													[(	byShrtAdr_Prim := 24, 
														byGrpAdr_Prim := 3, 
														eMod_Prim := E_DALIAddressType.Group, 
														byShrtAdr_Sec := 1, 
														byGrpAdr_Sec := 1, 
														//eMod_Sec := E_DALIAddressType.Short, 
														//byShrtAdr_Supl := 1,
														//eMod_Supl := E_DALIADDRESSTYPE.Group,
                                                        //byGrpAdr_Supl := 2, 
														DALI_LINE_NUM_PRIM := arrDALI_LINE_NUM_LIGHT[1], 
														DALI_LINE_NUM_SEC := 0, //0 = ingen zonestyring/vinduerække
														DALI_LINE_NUM_SUPL := arrDALI_LINE_NUM_PENDANTS[1]),
														
													(	byShrtAdr_Prim := 22, 
														byGrpAdr_Prim := 3, 
														eMod_Prim := E_DALIAddressType.Group, 
														byShrtAdr_Sec := 1, 
														byGrpAdr_Sec := 1, 
														//eMod_Sec := E_DALIAddressType.Short, 
														//byShrtAdr_Supl := 63, 
														DALI_LINE_NUM_PRIM := arrDALI_LINE_NUM_LIGHT[2], 
														DALI_LINE_NUM_SEC := 0, 
														DALI_LINE_NUM_SUPL := arrDALI_LINE_NUM_PENDANTS[2])];
														
	arrstLiveDataGruppe		: ARRAY [1..2] OF SH_Light.ST_LiveData;
	//stLiveData AT %MB22	: SH_Light.ST_LiveData;
	
	arrRunTuningGruppe: ARRAY[1..2] OF BOOL;
	
	bTopButtonZone1			: BOOL;
	bTopButtonZone1_Visu	: BOOL;
	bBottomButtonZone1		: BOOL;
	bBottomButtonZone1_Visu	: BOOL;
	bButtonZone2			: BOOL;
	bNeighborRoomsPir		: BOOL;
	fLuxOn					: REAL;
	fLuxDim					: REAL;
	tPIRDim					: TIME;
	tPIROff					: TIME;
	fOffsetSec				: REAL := 20;
	bOccupiedRoom			: BOOL;

	
// Sensor Settings
	//fbSensor					: SH_Light.FB_NIKO_P46xx_1Pcs;
	fbSensor					: SH_Light.FB_NIKO_P46xx_2Pcs;
	//bySensorAddr				: BYTE := x;
	arrSensorAddr				: ARRAY[1..2] OF BYTE := [3,4];
	bInitialize					: BOOL := TRUE;
	stDaliSensorSetup			: ST_DALI_NIKOP46SetupData := (
																nSensitivityPIRSegmentA := arrSensitivityOccupancy[1],
																nSensitivityPIRSegmentB := arrSensitivityOccupancy[2],
																nSensitivityPIRSegmentC := arrSensitivityOccupancy[3]);
	//bInitErr					: BOOL;
	//bInitDone					: BOOL;
	arrInitErr				: ARRAY [1..2] OF BOOL;
	arrInitDone				: ARRAY [1..2] OF BOOL;
	arrSensorScales				: ARRAY [1..10] OF SH_Light.ST_DALI_SensorScaleMode := [
																						(fMeassureMaxSensor := 1023, fReadMaxSensor := 1023),
																						(fMeassureMaxSensor := 1023, fReadMaxSensor := 1023),
																						8(())];
	bCancelHoldTimerOccupancy	: BOOL;
(*	eEventPriorityOccupancy		: E_DALIEventPriority := E_DALIEVENTPRIORITY.Middle;
	nHoldTimerOccupancy			: WORD := 5; // Value in s. 	
	nReportTimerOccupancy		: BYTE := 120; // Value in s, Preset manufacturer value
	nDeadtimeTimerOccupancy		: WORD := 100; // Value in ms, Predefined Value of DALI Standard
	bCancelHoldTimerOccupancy	: BOOL;
	nSensitivityOccupancy		: BYTE:= 3; //setting Sensivity (0..4) 0 (Off), 1 (Min), 2(Low), 3(High) and 4 (Max)

	bEnableLuxEvent				: BOOL;
	eEventPriorityBrightness	: E_DALIEventPriority := E_DALIEVENTPRIORITY.Middle;
	nDeadtimeTimerBrightness	: WORD := 1500; // Value in ms, Predefined Value of DALI Standard
	nHysteresisBrightness		: BYTE := 2; // Value in %
	nHysteresisMinBrightness	: BYTE := 10; // Absolute Value, depending on the manufacturer specific resolution
	nReportTimerBrightness		: BYTE := 120; // Value in s, Preset manufacturer value
*)

//ModbusComm setup
	
	fbWriteSPLuxLevel			: SH_Light.FB_TwoVal_SelectOne_RTrigChange;
	fbWritePirDelayTIme		: SH_Light.FB_TwoVal_SelectOne_RTrigChange;
	stRoomDataPLC				: SH_Light.ST_RoomDataPLC	:=	(
																	uiPirOffDelayTime	:= 30,
																	uiSpLuxLevel			:= 500,
																	uiPirDimDelayTime	:= 15,
																	uiSpDimLuxLevel		:= 200);
																	
	fbBallastOnHours			: SH_Light.FB_CountOnHours;
	bEnableHourCount			: BOOL := TRUE;
	
	//Non-persistent modbus data
	bPirActive_MB					AT%MX216.0	: BOOL;				//bPirLys i gammel kode
	uiActLuxLevel_MB			    AT%MB220		: UINT;				//intHMIAktueltLux i gammel kode
	uiActLightLevelPct_MB	        AT%MB224		: UINT;				//intDALI_Gruppe1_Lysniveau i gammel kode

	//For Conversion
	uiPirOffMinutes						: UINT;
	udTimeScaling						: UDINT := 60000;
	uiLuxOn								: UINT;
	
	//max values checks
	uiMaxLuxLevel						: UINT := 1023;
	uiMaxPirOffMinutes			     	: UINT := 180;
	
END_VAR

VAR CONSTANT
	//Sensor_DALI_LINE_NUM: BYTE := 3;
	Sensor_DALI_LINE_NUM				: BYTE := 2;
	arrDALI_LINE_NUM_LIGHT: ARRAY[1..2] OF BYTE := [1,2]; //korrekt rækkefølge nødvendig //rækkefølge og linje 
	arrDALI_LINE_NUM_PENDANTS: ARRAY[1..2] OF BYTE := [0,0]; //korrekt rækkefølge nødvendig. 0 = ingen pendler
	arrSensitivityOccupancy				: ARRAY[1..3] OF BYTE := [4,4,4];
END_VAR
VAR PERSISTENT
	stPirSensorData: SH_Light.ST_DALI_Sensor;
	arrstPirSensorDataLine: ARRAY[1..2] OF SH_Light.ST_DALI_Sensor; //hvad kan den her ??
	arrstTuneDataGruppe: ARRAY [1..2] OF SH_Light.ST_TuneData_EX;

	uiPirOffDelayTime_MB	AT%MB218	        : UINT;				//ntHMI_Pir_SetValue i gammel kode
	uiSPLuxLevel_MB			AT%MB222	   		: UINT;				//intHMI_Lux_SetValue i gammel kode
	uiBallastOnHours_MB		AT%MB226	        : UINT;		    	//dintHMILysbraendtimer1 i gammel kode
	byOnHoursOverflowCount			     		: BYTE;
END_VAR

A_Buttons();
A_LightCtrl();
A_Sensor();
A_ModbusComm();

ACTION A_Buttons:

bTopButtonZone1		:= bTopButtonZone1_Visu;
bBottomButtonZone1	:= bBottomButtonZone1_Visu;
END_ACTION

ACTION A_LightCtrl:
	

//gruppe 6
arrfbLysGruppe[1]( 
	nZoneID:= 1, 
	bButtonZone1:= bTopButtonZone1,
	bBottomButtonZone1 := bBottomButtonZone1, 
	bButtonZone2:= bButtonZone2,
	fLuxOn:= fLuxOn, 
	fLuxDim:= fLuxDim, 
	tPIRDim:= tPIRDim, 
	tPIROff:= tPIROff, 
	fOffsetSec:= fOffsetSec, 
	bReInit:= , 
	stDaliSetup:= arrstDaliSetupGruppe[1], 
	ipCommunication_Prim:= P_DALI_Background.arrfbKL6821Communication[arrDALI_LINE_NUM_LIGHT[1]], 
	//ipCommunication_Sec:= P_DALI_Background.arrfbKL6821Communication[arrDALI_LINE_NUM_LIGHT[1]], //samme som lyslinjen, hvis den ikke eksisterer
	//ipCommunication_Supl:= P_DALI_Background.arrfbKL6821Communication[arrDALI_LINE_NUM_LIGHT[1]],//samme som lyslinjen, hvis den ikke eksisterer 
	fMinOutputPowerLevelRoom:= 15, 
	fMaxOutputPowerLevelRoom:= 100, 
	nCycleTimeInMS:= SH_Light.DALI_Param.nPlcTaskCycleTimeInMS*nDimCmdCycleTimeFactor , 
	bRunTuning:= arrRunTuningGruppe[1], 
	bOccupiedRoom=> , 
	bError_Prim=> , 
	nError_Prim=> , 
	stTuneData:=arrstTuneDataGruppe[1] , 
	stPirSensorData:= stPirSensorData, 					//samme sensordata
	stLiveData:= arrstLiveDataGruppe[1]);

//gruppe 15	
arrfbLysGruppe[2]( 
	nZoneID:= 1, 
	bButtonZone1:= bTopButtonZone1,
	bBottomButtonZone1 := bBottomButtonZone1, 
	bButtonZone2:= bButtonZone2,
	fLuxOn:= fLuxOn, 
	fLuxDim:= fLuxDim, 
	tPIRDim:= tPIRDim, 
	tPIROff:= tPIROff, 
	fOffsetSec:= fOffsetSec, 
	bReInit:= , 
	stDaliSetup:= arrstDaliSetupGruppe[2], 
	ipCommunication_Prim:= P_DALI_Background.arrfbKL6821Communication[arrDALI_LINE_NUM_LIGHT[2]], 
	//ipCommunication_Sec:= P_DALI_Background.arrfbKL6821Communication[arrDALI_LINE_NUM_LIGHT[2]], //samme som lyslinjen, hvis den ikke eksisterer
	//ipCommunication_Supl:= P_DALI_Background.arrfbKL6821Communication[arrDALI_LINE_NUM_LIGHT[2]], //samme som lyslinjen, hvis den ikke eksisterer 
	fMinOutputPowerLevelRoom:= 15, 
	fMaxOutputPowerLevelRoom:= 100, 
	nCycleTimeInMS:= SH_Light.DALI_Param.nPlcTaskCycleTimeInMS*nDimCmdCycleTimeFactor , 
	bRunTuning:= arrRunTuningGruppe[2], 
	bOccupiedRoom=> , 
	bError_Prim=> , 
	nError_Prim=> , 
	stTuneData:=arrstTuneDataGruppe[2] , 
	stPirSensorData:= stPirSensorData, 					//samme sensordata
	stLiveData:= arrstLiveDataGruppe[2]);
END_ACTION

ACTION A_ModbusComm:
//Manage data for modbus communication

//Manage data for read-only in PLC
stRoomDataPLC.bPirActive			:= stPirSensorData.bPrc;
stRoomDataPLC.uiActLuxLevel			:= TO_UINT(TRUNC(stPirSensorData.fBrightness));
stRoomDataPLC.uiActLightLevelPct	:= TO_UINT(TRUNC(arrfbLysGruppe[1].fbBallast.fActlLgtLvl_Prim));
		//stRoomDataPLC.uiActLightLevelPct	:= TO_UINT(TRUNC(fbLys.fbBallast.fActlLgtLvl_Prim)); //if only one group light control
stRoomDataPLC.uiBallastOnHours		:= uiBallastOnHours_MB; //The calculation for BallastOnHours is stored directly to the MB register below


//Assign data for read-only to MB registers
bPirActive_MB			:= stRoomDataPLC.bPirActive;
uiActLuxLevel_MB		:= stRoomDataPLC.uiActLuxLevel;
uiActLightLevelPct_MB	:= stRoomDataPLC.uiActLightLevelPct;

	//calculate BallastOnHours
	fbBallastOnHours(
		bEnableHourCount	:= bEnableHourCount,
		bPauseCount			:= arrfbLysGruppe[1].fbLightCtrl.bOffZone1,
		uiOnHours			:= uiBallastOnHours_MB,			//OnHours is updated here
		byOverflowCount		:= byOnHoursOverflowCount);


//Manage data for read/write for both PLC and MB registers
fbWriteSPLuxLevel(	nMaxValOut	:= uiMaxLuxLevel,
					nValIn1		:= uiSPLuxLevel_MB,		//nValIn1 takes priotity in case of download or restart
					nValIn2		:= stRoomDataPLC.uiSpLuxLevel,
					nValOut		=> uiLuxOn
				);


fbWritePirDelayTIme(	nMaxValOut	:= uiMaxPirOffMinutes,
						nValIn1		:= uiPirOffDelayTime_MB,		//nValIn1 takes priotity in case of download or restart
						nValIn2		:= stRoomDataPLC.uiPirOffDelayTime,
						nValOut		=> uiPirOffMinutes
					);
					

//Convert read/write modbus data to appropriate datatypes in PLC
fLuxOn	:= TO_REAL(uiLuxOn);			
tPIROff	:= TO_TIME(uiPirOffMinutes*udTimeScaling); //Time conversion defaults to ms

fLuxDim	:= TO_REAL(stRoomDataPLC.uiSpDimLuxLevel);			
tPIRDim	:= TO_TIME(stRoomDataPLC.uiPirDimDelayTime*udTimeScaling); //Time conversion defaults to ms
END_ACTION

ACTION A_Sensor:

fbSensor.ipCommunication := P_DALI_Background.arrfbKL6821Communication[Sensor_DALI_LINE_NUM];

(*
fbSensor(
	byShrtAdr:= bySensorAddr,
	bInitialize:= bInitialize, 
	DALI_LINE_NUM:= Sensor_DALI_LINE_NUM, 
 	//bCancelHoldTimerOccupancy:= bCancelHoldTimerOccupancy, 
	stSensorSetup := stDaliSensorSetup,
	bInitErr=> bInitErr, 
	bInitDone=> bInitDone,
	stPirSensorData:= stPirSensorData, 
	arrSensorScales:= arrSensorScales);
*)

fbSensor(
	arrShrtAdr:= arrSensorAddr,
	bInitialize:= bInitialize, 
	DALI_LINE_NUM:= Sensor_DALI_LINE_NUM, 
 	//bCancelHoldTimerOccupancy:= bCancelHoldTimerOccupancy, 
	stSensorSetup := stDaliSensorSetup,
	arrInitErr=> arrInitErr, 
	arrInitDone=> arrInitDone,
	stPirSensorData:= stPirSensorData, 
	arrSensorScales:= arrSensorScales);
END_ACTION

END_PROGRAM

// ---- POUs/Alle_Rum/Trapper/P_Trappe_T5.TcPOU
PROGRAM P_Trappe_T5
VAR
	bDigitalPir				AT%I*	: BOOL;
	bTrappelysNC		AT%Q*	: BOOL;
	
	fbTon_Off				: TON;
	tPirTidOff				: TIME;
	tPirTidOff_PLC	: TIME := T#1M;
	bIngenAktivitet		: BOOL;
	bTrappeLys			: BOOL;
	
	//Modbus data Read
	bTrappeAktivitet		: BOOL;
	//Modbus data Read/Wrtite
	bPirTidOff_MB			: TIME;
	
END_VAR


bIngenAktivitet	:= NOT bDigitalPir;
tPirTidOff		:= tPirTidOff_PLC;

fbTon_Off(IN:= bIngenAktivitet, PT:= tPirTidOff);

IF bDigitalPir  THEN
	bTrappeLys := TRUE;
END_IF
IF fbTon_Off.Q THEN
	bTrappeLys := FALSE;
END_IF

bTrappelysNC 	:= NOT bTrappeLys;

END_PROGRAM

// ---- POUs/EnOcean/P_EnOcean.TcPOU
PROGRAM P_EnOcean
VAR
	fbKL6581			: FB_KL6581;
	stKL6581_in  AT %I* : KL6581_INPUT;
	stKL6581_out AT %Q*	: KL6581_OUTPUT;
	stKL6581			: STR_KL6581;
	bInitCom			: BOOL := TRUE;
	
	arrEnOcean_Search	: ARRAY [1..8] OF FB_EnOcean_Search;
	nSearchIdx			: BYTE;
	bSerach				: BOOL;
	arrDevices			: ARRAY [1..8] OF INT;
	arrID				: ARRAY [1..8, 0..255] OF DWORD;
	
		//Trykknapper Atrium
	fbAtriumNiveau_Tryk_PladeB				: FB_Rec_RPS_Switch;
	fbAtriumNiveau_Tryk_Sevice				: FB_Rec_RPS_Switch;			

	//Trykknapper på gange

	
	//Trykknapper i rum
fbRum_1_111_Tryk						: FB_Rec_RPS_Switch;

END_VAR

VAR CONSTANT
	byNode_1: BYTE := 1;
	byNode_2: BYTE := 2;
	byNode_3: BYTE := 3;
	byNode_4: BYTE := 4;
	byNode_5: BYTE := 5;
	byNode_6: BYTE := 6;
	byNode_7: BYTE := 7;
	byNode_8: BYTE := 8;
END_VAR


(* Kommunikation mit der KL6581. *)
(* Communication with the KL6581. *)
fbKL6581(
	bInit			:= bInitCom,
	nIdx			:= 2,
	stKL6581_in		:= stKL6581_In,
	stKL6581_out	:= stKL6581_Out,
	bReady			=> ,
	bBusy			=> ,
	bError			=> ,
	iErrorID		=> ,
	str_KL6581		=> stKL6581);

GVL_AHDataModbus.EnOceanError	:= TO_UINT(fbKL6581.iErrorID);
(* Warten bis der Kommunikationsbaustein initialisiert wurde.*)
(* Wait until the communication function block has been initialized. *)
IF (NOT fbKL6581.bReady) THEN
	RETURN;
END_IF

FOR nSearchIdx:= 1 TO 8 DO
	arrEnOcean_Search[nSearchIdx](
		bStart:= TRUE, 
		str_KL6581:= stKL6581 , 
		byNode:= nSearchIdx, 
		bReceive=> , 
		iDevices=>arrDevices[nSearchIdx] , 
		ar_ID=> );
		
		MEMCPY(ADR(arrID[nSearchIdx,0]), ADR(arrEnOcean_Search[nSearchIdx].ar_ID), SIZEOF(arrEnOcean_Search[nSearchIdx].ar_ID)); 
END_FOR

//Gange



//RUM
 //
P_Rum_1_111();

//AtriumNiveau
A_AtriumNiveau();

ACTION A_AtriumNiveau:
fbAtriumNiveau_Tryk_PladeB(
	str_KL6581:=stKL6581 , 
	byNode:=0, 
	dw_ID:= 16#0029B92D, 
	str_EnOceanSwitch=> GVL_EnOcean.strEnOceanSwitch_AtriumNiveau_PladeB,
	by_Node=> , 
	bReceive=> );

//knap 2 
(*
fbAtriumNiveau_Tryk_Sevice(
	str_KL6581:=stKL6581 , 
	byNode:=0, 
	dw_ID:= 16#00FEE4FE87, 
	str_EnOceanSwitch=> GVL_EnOcean.strEnOceanSwitch_AtriumNiveau_Service, 
	by_Node=> , 
	bReceive=> );
*)


//Den rigtigt: 16#0029B92D
END_ACTION

ACTION P_Rum_1_111:
fbRum_1_111_Tryk(
	str_KL6581:=stKL6581 , 
	byNode:=0 , 
	dw_ID:=  16#0029ABB1, 
	str_EnOceanSwitch=> GVL_EnOcean.strEnOceanSwitch_Rum_1_111, 
	by_Node=> , 
	bReceive=> );
	
fbRum_1_111_Tryk(
	str_KL6581:=stKL6581 , 
	byNode:=0 , 
	dw_ID:=  16#0029AB7A, 
	str_EnOceanSwitch=> GVL_EnOcean.strEnOceanSwitch_Rum_1_111, 
	by_Node=> , 
	bReceive=> );
END_ACTION

ACTION P_Rum_5_454:
(*fbRum_5_454_Tryk(
	str_KL6581:=stKL6581 , 
	byNode:=4 , 
	dw_ID:=  16#0029B75D, 
	str_EnOceanSwitch=> GVL_EnOcean.strEnOceanSwitch_Rum_5_454, 
	by_Node=> , 
	bReceive=> );
*)
END_ACTION

END_PROGRAM

// ---- VISUs/MAIN.TcPOU
PROGRAM MAIN
VAR
	nAlive: INT;
	breset: BOOL;
	nDemoVariable : INT;
	nCX8200_State	AT %I*	: UINT;
	P_Rum_6_217: INT;
END_VAR

VAR PERSISTENT
	nDemoVar_Persist: INT;
END_VAR

nAlive:= nAlive + 1;
GVL_AHDataModbus.nCX8200_State_MB := nCX8200_State;

P_SystemDK.M_nCyclic(bReset := breset );
P_DALI_DIAG();
DALI_Commissioning();
P_DALI_Energy_Line();
P_AHModbusComm();


//Gange
P_Gang_2_546A();
P_Gang_3_545();
P_Gang_3_558();
P_gang_7_501();
//Rum


//FoldeDøre
//P_Foldedoer_5_125();



//Testprogrammer
//P_DALI_Energy_Firmware_Test();

END_PROGRAM

// ---- POUs/Alle_Rum/Gange/Gang_1_5_441/Visualization_4_330_1_1_1_1_2_2.TcVIS
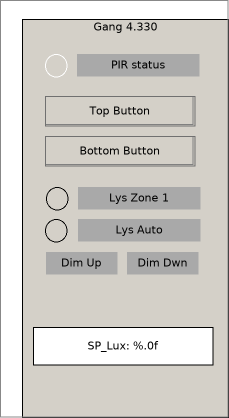
VISUALIZATION Visualization_4_330_1_1_1_1_2_2  // 229x418
    RoundedRectangle (22,19 207x399), "Gang 4.330"
    Rectangle (33,327 180x38), "SP_Lux: %.0f", text variable: P_Gang_5_135A.arrfbLysGruppe[1].fbLightCtrl.fLuxZone1
    Button (45,96 150x30), "Top Button"
        tap P_Gang_5_135A.bTopButtonZone1_Visu
    Button (45,136 150x30), "Bottom Button"
        tap P_Gang_5_135A.bBottomButtonZone1_Visu
    Ellipse (46,187 22x23), colour toggle: P_Gang_5_135A.fbLys.fbLightCtrl.bOnZone1
    Rectangle (78,187 122x22), "Lys Zone 1"
    Rectangle (46,252 71x22), "Dim Up", colour toggle: P_Gang_5_135A.arrfbLysGruppe[1].fbLightCtrl.bDimUp
    Rectangle (127,252 71x22), "Dim Dwn", colour toggle: P_Gang_5_135A.arrfbLysGruppe[1].fbLightCtrl.bDimDwn
    Ellipse (45,219 22x23), colour toggle: P_Gang_5_135A.arrfbLysGruppe[1].fbLightCtrl.bAutoZone1
    Rectangle (78,219 122x22), "Lys Auto"
    Ellipse (45,54 22x23), colour toggle: P_Gang_5_135A.arrfbLysGruppe[1].fbLightCtrl.bPIR
    Rectangle (77,54 122x22), "PIR status"
END_VISUALIZATION

// ---- POUs/Alle_Rum/Gange/Gang_7_501/Visualization_4_330.TcVIS
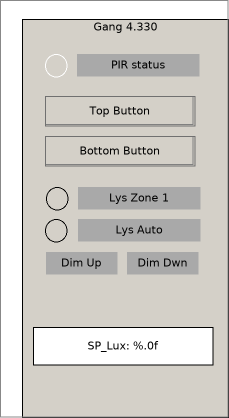
VISUALIZATION Visualization_4_330  // 229x418
    RoundedRectangle (22,19 207x399), "Gang 4.330"
    Rectangle (33,327 180x38), "SP_Lux: %.0f", text variable: P_Gang_2_143A.arrfbLysGruppe[1].fbLightCtrl.fLuxZone1
    Button (45,96 150x30), "Top Button"
        tap P_Gang_2_143A.bTopButtonZone1_Visu
    Button (45,136 150x30), "Bottom Button"
        tap P_Gang_2_143A.bBottomButtonZone1_Visu
    Ellipse (46,187 22x23), colour toggle: P_Gang_2_143A.fbLys.fbLightCtrl.bOnZone1
    Rectangle (78,187 122x22), "Lys Zone 1"
    Rectangle (46,252 71x22), "Dim Up", colour toggle: P_Gang_2_143A.arrfbLysGruppe[1].fbLightCtrl.bDimUp
    Rectangle (127,252 71x22), "Dim Dwn", colour toggle: P_Gang_2_143A.arrfbLysGruppe[1].fbLightCtrl.bDimDwn
    Ellipse (45,219 22x23), colour toggle: P_Gang_2_143A.arrfbLysGruppe[1].fbLightCtrl.bAutoZone1
    Rectangle (78,219 122x22), "Lys Auto"
    Ellipse (45,54 22x23), colour toggle: P_Gang_2_143A.arrfbLysGruppe[1].fbLightCtrl.bPIR
    Rectangle (77,54 122x22), "PIR status"
END_VISUALIZATION

// ---- POUs/Alle_Rum/Gange/Gang_3_558/Visualization_4_330_3.TcVIS
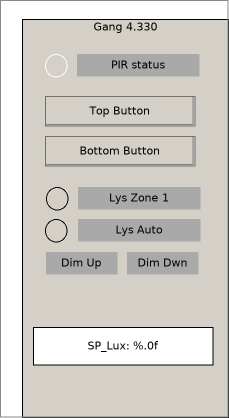
VISUALIZATION Visualization_4_330_3  // 229x418
    RoundedRectangle (22,19 207x399), "Gang 4.330"
    Rectangle (33,327 180x38), "SP_Lux: %.0f", text variable: P_Gang_2_143A.arrfbLysGruppe[1].fbLightCtrl.fLuxZone1
    Button (45,96 150x30), "Top Button"
        tap P_Gang_2_143A.bTopButtonZone1_Visu
    Button (45,136 150x30), "Bottom Button"
        tap P_Gang_2_143A.bBottomButtonZone1_Visu
    Ellipse (46,187 22x23), colour toggle: P_Gang_2_143A.fbLys.fbLightCtrl.bOnZone1
    Rectangle (78,187 122x22), "Lys Zone 1"
    Rectangle (46,252 71x22), "Dim Up", colour toggle: P_Gang_2_143A.arrfbLysGruppe[1].fbLightCtrl.bDimUp
    Rectangle (127,252 71x22), "Dim Dwn", colour toggle: P_Gang_2_143A.arrfbLysGruppe[1].fbLightCtrl.bDimDwn
    Ellipse (45,219 22x23), colour toggle: P_Gang_2_143A.arrfbLysGruppe[1].fbLightCtrl.bAutoZone1
    Rectangle (78,219 122x22), "Lys Auto"
    Ellipse (45,54 22x23), colour toggle: P_Gang_2_143A.arrfbLysGruppe[1].fbLightCtrl.bPIR
    Rectangle (77,54 122x22), "PIR status"
END_VISUALIZATION

// ---- POUs/Alle_Rum/Gange/Gang_Atrium/Visualization_5_338_2.TcVIS
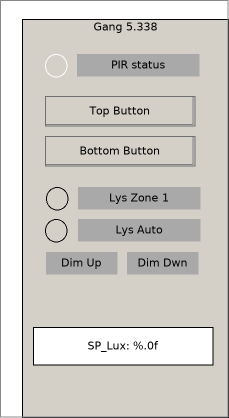
VISUALIZATION Visualization_5_338_2  // 229x418
    RoundedRectangle (22,19 207x399), "Gang 5.338"
    Rectangle (33,327 180x38), "SP_Lux: %.0f", text variable: P_Gang_5_338.arrfbLysGruppe[1].fbLightCtrl.fLuxZone1
    Button (45,96 150x30), "Top Button"
        tap P_Gang_5_338.bTopButtonZone1_Visu
    Button (45,136 150x30), "Bottom Button"
        tap P_Gang_5_338.bBottomButtonZone1_Visu
    Ellipse (46,187 22x23), colour toggle: P_Gang_5_338.arrfbLysGruppe[1].fbLightCtrl.bOnZone1
    Rectangle (78,187 122x22), "Lys Zone 1"
    Rectangle (46,252 71x22), "Dim Up", colour toggle: P_Gang_5_338.arrfbLysGruppe[1].fbLightCtrl.bDimUp
    Rectangle (127,252 71x22), "Dim Dwn", colour toggle: P_Gang_5_338.arrfbLysGruppe[1].fbLightCtrl.bDimDwn
    Ellipse (45,219 22x23), colour toggle: P_Gang_5_338.arrfbLysGruppe[1].fbLightCtrl.bAutoZone1
    Rectangle (78,219 122x22), "Lys Auto"
    Ellipse (45,54 22x23), colour toggle: P_Gang_5_338.arrfbLysGruppe[1].fbLightCtrl.bPIR
    Rectangle (77,54 122x22), "PIR status"
END_VISUALIZATION

// ---- POUs/Alle_Rum/Rum_Med_DALI_Pir/1_Rum_5_125_Og_5_127_Foldedoer/Visualization_5_352_1_1_1_1_1_1.TcVIS
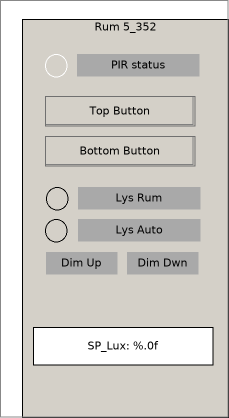
VISUALIZATION Visualization_5_352_1_1_1_1_1_1  // 229x418
    RoundedRectangle (22,19 207x399), "Rum 5_352"
    Rectangle (33,327 180x38), "SP_Lux: %.0f", text variable: P_Rum_4_324.fbLys.fbLightCtrl.fLuxZone1
    Button (45,96 150x30), "Top Button"
        tap P_Rum_5_352.bTopButtonZone1_Visu
    Button (45,136 150x30), "Bottom Button"
        tap P_Rum_5_352.bBottomButtonZone1_Visu
    Ellipse (46,187 22x23), colour toggle: P_Rum_5_352.fbLys.fbLightCtrl.bOnZone1
    Rectangle (78,187 122x22), "Lys Rum"
    Rectangle (46,252 71x22), "Dim Up", colour toggle: P_Rum_5_352.fbLys.fbLightCtrl.bDimUp
    Rectangle (127,252 71x22), "Dim Dwn", colour toggle: P_Rum_5_352.fbLys.fbLightCtrl.bDimDwn
    Ellipse (45,219 22x23), colour toggle: P_Rum_5_352.fbLys.fbLightCtrl.bAutoZone1
    Rectangle (78,219 122x22), "Lys Auto"
    Ellipse (45,54 22x23), colour toggle: P_Rum_5_352.fbLys.fbLightCtrl.bPIR
    Rectangle (77,54 122x22), "PIR status"
END_VISUALIZATION

// ---- POUs/Alle_Rum/Rum_Med_DALI_Pir/Rum_5_456/Visualization_4_330_1_1_1_1_2_1_1_1_3_1_1_1_1_1.TcVIS
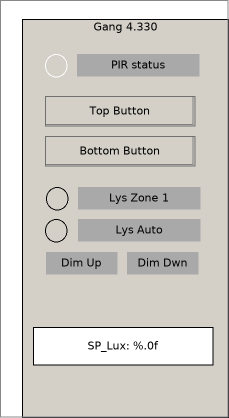
VISUALIZATION Visualization_4_330_1_1_1_1_2_1_1_1_3_1_1_1_1_1  // 229x418
    RoundedRectangle (22,19 207x399), "Gang 4.330"
    Rectangle (33,327 180x38), "SP_Lux: %.0f", text variable: P_Gang_5_135A.arrfbLysGruppe[1].fbLightCtrl.fLuxZone1
    Button (45,96 150x30), "Top Button"
        tap P_Gang_5_135A.bTopButtonZone1_Visu
    Button (45,136 150x30), "Bottom Button"
        tap P_Gang_5_135A.bBottomButtonZone1_Visu
    Ellipse (46,187 22x23), colour toggle: P_Gang_5_135A.fbLys.fbLightCtrl.bOnZone1
    Rectangle (78,187 122x22), "Lys Zone 1"
    Rectangle (46,252 71x22), "Dim Up", colour toggle: P_Gang_5_135A.arrfbLysGruppe[1].fbLightCtrl.bDimUp
    Rectangle (127,252 71x22), "Dim Dwn", colour toggle: P_Gang_5_135A.arrfbLysGruppe[1].fbLightCtrl.bDimDwn
    Ellipse (45,219 22x23), colour toggle: P_Gang_5_135A.arrfbLysGruppe[1].fbLightCtrl.bAutoZone1
    Rectangle (78,219 122x22), "Lys Auto"
    Ellipse (45,54 22x23), colour toggle: P_Gang_5_135A.arrfbLysGruppe[1].fbLightCtrl.bPIR
    Rectangle (77,54 122x22), "PIR status"
END_VISUALIZATION

// ---- POUs/DALI/DALI_Setup/VISUs/Visu_DALICommissioning/Visu_KL6821Configuration.TcVIS
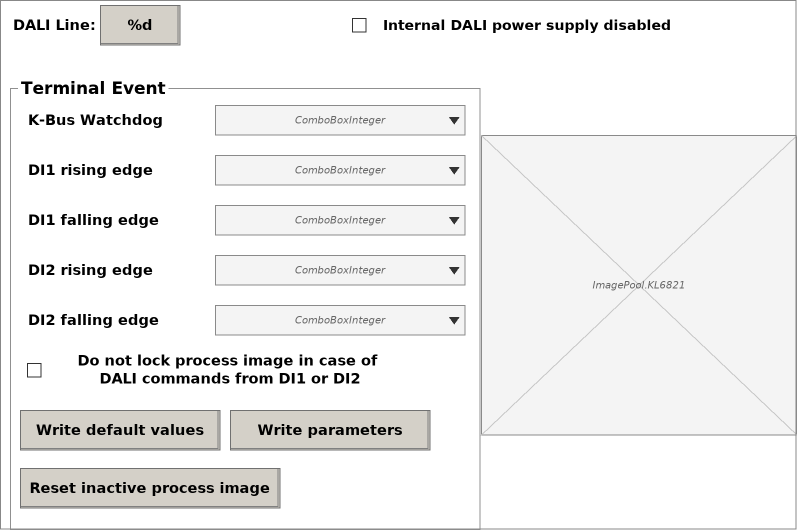
VISUALIZATION Visu_KL6821Configuration  // 797x530
    GroupBox (10,80 470x450), "Terminal Event"
        Textfield (15,25 170x30), "K-Bus Watchdog"
        ComboBoxInteger (205,25 250x30), variable: P_DALI_Background.eCommandKBusWatchdog, text list: 'CommandOnTerminalEvent'
        Textfield (15,75 170x30), "DI1 rising edge"
        Textfield (15,125 170x30), "DI1 falling edge"
        ComboBoxInteger (205,75 250x30), variable: P_DALI_Background.eCommandDI1RisingEdge, text list: 'CommandOnTerminalEvent'
        ComboBoxInteger (205,125 250x30), variable: P_DALI_Background.eCommandDI1FallingEdge, text list: 'CommandOnTerminalEvent'
        Textfield (15,175 170x30), "DI2 rising edge"
        ComboBoxInteger (205,175 250x30), variable: P_DALI_Background.eCommandDI2RisingEdge, text list: 'CommandOnTerminalEvent'
        Textfield (15,225 170x30), "DI2 falling edge"
        ComboBoxInteger (205,225 250x30), variable: P_DALI_Background.eCommandDI2FallingEdge, text list: 'CommandOnTerminalEvent'
        Button (220,330 200x40), "Write parameters"
            OnMouseClick: execute { P_DALI_Background.bInitialize := TRUE; }
        Button (10,330 200x40), "Write default values"
            OnMouseClick: execute { P_DALI_Background.bDefaultValues := TRUE; }
        Button (10,388 260x40), "Reset inactive process image"
            OnMouseClick: execute { P_DALI_Background.bResetInactiveProcessImage := TRUE; }
        Checkbox (15,275 35x30), variable: P_DALI_Background.bDoNotLockProcessImage
        Textfield (50,267 340x45), "Do not lock process image in case of DALI commands from DI1 or DI2"
    Image (481,135 316x300), image: ImagePool.KL6821
    Group (350,10 330x30)
        Checkbox (0,0 34x30), variable: P_DALI_Background.bInternalPowerSupplyDisabled
        Textfield (30,0 294x30), "Internal DALI power supply disabled"
    Group (10,5 170x40)
        Textfield (0,0 110x40), "DALI Line:"
        Button (90,0 80x40), "%d", text variable: GVL_Internal.nDALILine
            OnMouseClick: write the text variable via Default, min 1, max 10, title "Choose line"
END_VISUALIZATION

// ---- POUs/DALI/DALI_Setup/VISUs/Visu_DALICommissioning/Visu_Part103MemoryBank.TcVIS
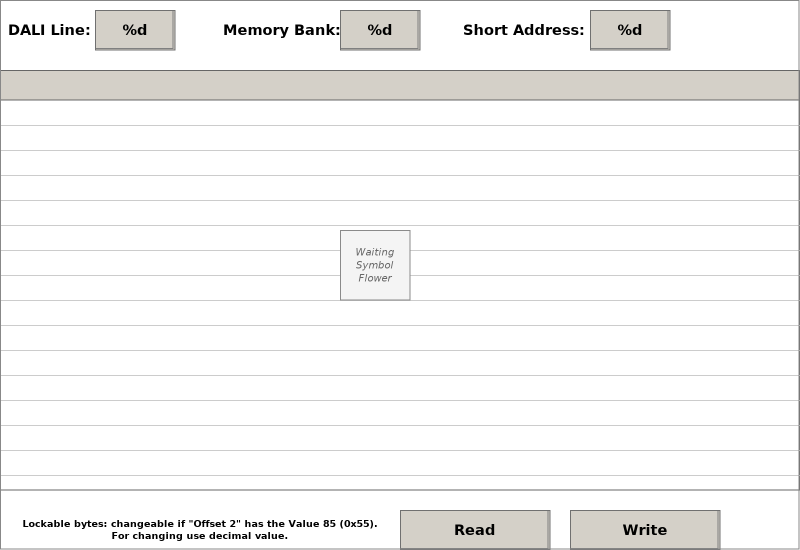
VISUALIZATION Visu_Part103MemoryBank  // 800x550
    Table (0,70 800x420), data array: DALI_Commissioning.fbPart103MemoryPages.aMemoryBank
        p3854506369: DALI_Commissioning.fbPart103MemoryPages.aMemoryBank[INDEX].sOffset
        p1892666644: DALI_Commissioning.fbPart103MemoryPages.aMemoryBank[INDEX].sName
        p338671338: DALI_Commissioning.fbPart103MemoryPages.aMemoryBank[INDEX].nValueDec
        p2170511999: DALI_Commissioning.fbPart103MemoryPages.aMemoryBank[INDEX].nValueHex
        p1755163831: Value Dec
        p4092479075: Value Hex
        p1137915858: DALI_Commissioning.fbPart103MemoryPages.nOffset
        Columns.Column.[0].Template: DALI_Commissioning.fbPart103MemoryPages.aNoValue[INDEX]
        Columns.Column.[1].Template: DALI_Commissioning.fbPart103MemoryPages.aNoValue[INDEX]
        Columns.Column.[2].Template: DALI_Commissioning.fbPart103MemoryPages.aNoValue[INDEX]; DALI_Commissioning.fbPart103MemoryPages.nMemoryBank=0; OnMouseClick: write the text variable via Default, min 0, max 255, title "Lockable variable decimal"
        Columns.Column.[3].Template: DALI_Commissioning.fbPart103MemoryPages.aNoValue[INDEX]; OnMouseClick: write the text variable via Default, title "Lockable variable hexadecimal"
    Button (400,510 150x40), "Read"
        OnMouseClick: execute { DALI_Commissioning.fbPart103MemoryPages.bRead := TRUE; }
    Button (570,510 150x40), "Write"
        OnMouseClick: execute { DALI_Commissioning.fbPart103MemoryPages.bWrite := TRUE; }
    Textfield (15,510 370x40), "Lockable bytes: changeable if "Offset 2" has the Value 85 (0x55). For changing use decimal value."
    WaitingSymbolFlower (340,230 70x70), invisible if: DALI_Commissioning.fbPart103MemoryPages.bHideWaitSymbol
    Textfield (460,10 130x40), "Short Address:"
    Button (590,10 80x40), "%d", text variable: DALI_Commissioning.fbPart103MemoryPages.nAddress
        OnMouseClick: write the text variable via Default, min 0, max 63, title "Insert Short Address"
    Group (220,10 200x40)
        Textfield (0,0 150x40), "Memory Bank:"
        Button (120,0 80x40), "%d", text variable: DALI_Commissioning.fbPart103MemoryPages.nMemoryBank
            OnMouseClick: write the text variable via Default, min 0, max 255, title "Insert Memory Bank"
    Group (5,10 170x40)
        Textfield (0,0 110x40), "DALI Line:"
        Button (90,0 80x40), "%d", text variable: GVL_Internal.nDALILine
            OnMouseClick: write the text variable via Default, min 1, max 10, title "Choose line"
END_VISUALIZATION

// ---- POUs/DALI/DALI_Setup/VISUs/Visu_DALICommissioning/Visu_Part207Parameters.TcVIS
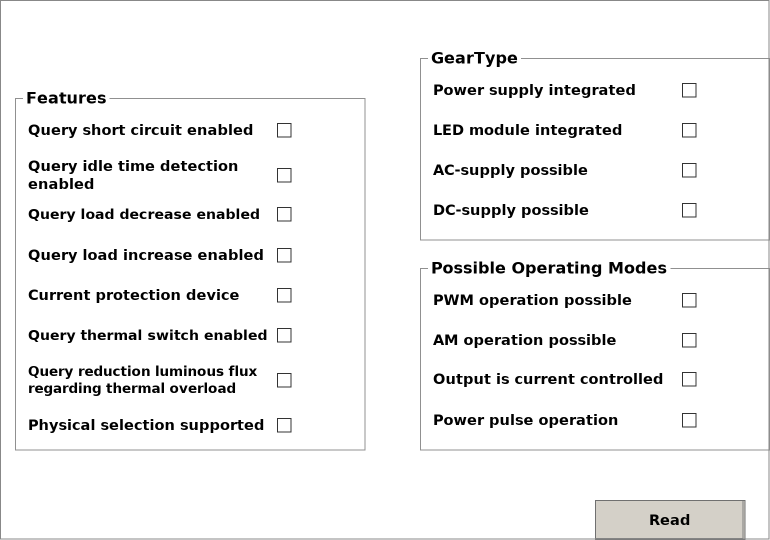
VISUALIZATION Visu_Part207Parameters  // 770x540
    Button (595,500 150x40), "Read"
        OnMouseClick: execute { DALI_Commissioning.fbPart207LED.bReadParameter:=TRUE; }
    GroupBox (420,50 350x190), "GearType"
        Textfield (10,25 220x30), "Power supply integrated"
        Checkbox (260,25 30x30), variable: DALI_Commissioning.fbPart207LED.bLEDPowerSupply, input disabled if: True
        Textfield (10,65 220x30), "LED module integrated"
        Textfield (10,145 220x30), "DC-supply possible"
        Textfield (10,105 220x30), "AC-supply possible"
        Checkbox (260,65 30x30), variable: DALI_Commissioning.fbPart207LED.bLEDModule, input disabled if: True
        Checkbox (260,145 30x30), variable: DALI_Commissioning.fbPart207LED.bDCSupply, input disabled if: True
        Checkbox (260,105 30x30), variable: DALI_Commissioning.fbPart207LED.bACSupply, input disabled if: True
    GroupBox (15,90 350x360), "Features"
        Textfield (10,25 240x30), "Query short circuit enabled"
        Checkbox (260,25 30x30), variable: DALI_Commissioning.fbPart207LED.bQueryShortCircuitEnabled, input disabled if: True
        Textfield (10,65 240x40), "Query idle time detection enabled"
        Textfield (10,150 240x30), "Query load increase enabled"
        Textfield (10,109 240x30), "Query load decrease enabled"
        Checkbox (260,70 30x30), variable: DALI_Commissioning.fbPart207LED.bQueryIdleTimeDetectionEnabled, input disabled if: True
        Checkbox (260,150 30x30), variable: DALI_Commissioning.fbPart207LED.bQueryLoadIncreaseEnabled, input disabled if: True
        Checkbox (260,109 30x30), variable: DALI_Commissioning.fbPart207LED.bQueryLoadDecreaseEnabled, input disabled if: True
        Textfield (10,190 240x30), "Current protection device"
        Checkbox (260,190 30x30), variable: DALI_Commissioning.fbPart207LED.bQueryCurrentProtectionDevicePresent, input disabled if: True
        Checkbox (260,230 30x30), variable: DALI_Commissioning.fbPart207LED.bQueryThermalSwitchEnabled, input disabled if: True
        Checkbox (260,275 30x30), variable: DALI_Commissioning.fbPart207LED.bQueryReductionOfLuminouFluxRegardingThermalOverloadEnabled, input disabled if: True
        Checkbox (260,320 30x30), variable: DALI_Commissioning.fbPart207LED.bPhysicalSelectionSupported, input disabled if: True
        Textfield (10,230 240x30), "Query thermal switch enabled"
        Textfield (10,270 240x40), "Query reduction luminous flux regarding thermal overload"
        Textfield (10,320 240x30), "Physical selection supported"
    GroupBox (420,260 350x190), "Possible Operating Modes", invisible if: DALI_Commissioning.fbPart207LED.bInvisible
        Checkbox (260,25 30x30), variable: DALI_Commissioning.fbPart207LED.bPWMOperation, input disabled if: True
        Textfield (10,65 240x30), "AM operation possible"
        Textfield (10,145 240x30), "Power pulse operation"
        Textfield (10,104 240x30), "Output is current controlled"
        Checkbox (260,65 30x30), variable: DALI_Commissioning.fbPart207LED.bAMOperation, input disabled if: True
        Checkbox (260,145 30x30), variable: DALI_Commissioning.fbPart207LED.bPowerPulseOperation, input disabled if: True
        Checkbox (260,104 30x30), variable: DALI_Commissioning.fbPart207LED.bOutputCurrentControlled, input disabled if: True
        Textfield (10,25 240x30), "PWM operation possible"
END_VISUALIZATION
